ABB RobotStudio station: RoboX0.rspag

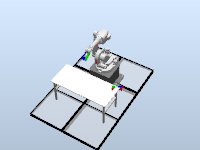
--- station ---
Station RoboX0 (saved by RobotStudio 21.3.9676.1)
Controller IRB1600_10_145, task T_ROB1: task frame (RAPID world) sits at (0, 0, 520) mm in the station
Controller IRB1600_10_145
  mechanical unit ROB_1: IRB1600_10_145__01_2, 6 joints, base frame (0, 0, 0) mm
Layout (positions relative to the parent item):
  - IRB1600_10_145__01_2 [mechanism, from Robots\IRB1600_10_145_G_01.rslib] at (0, 0, 520) mm; joint values [0, 0, 0, 0, 0.5236, 0] (rad or m)
  - подставка [part, from Libraries\box.rslib]
  - Стол сборка_4 [part, from Libraries\table.rslib] at (975, 0, 0) mm, rotated rx 0 ry 0 rz 90 deg
  - gripper2 [mechanism, from Libraries\gripper.rslib] at (806.29, 0, 1674) mm, rotated rx 180 ry 60 rz 180 deg; joint values [0] (rad or m)
Attachment: gripper2 is attached to IRB1600_10_145__01_2 / Link6

--- Backups/IRB1600_10_145/RAPID/TASK1/PROGMOD/CalibData.mod ---
MODULE CalibData
    TASK PERS wobjdata Workobject_1:=[FALSE,TRUE,"",[[606.263,790,210],[0.707106781,0,0,0.707106781]],[[-100,-100,0],[0,-0.707106781,0.707106781,0]]];
    PERS tooldata gripper:=[TRUE,[[0,0,115],[1,0,0,0]],[0.5,[0,0,30],[1,0,0,0],0,0,0]];
ENDMODULE

--- Backups/IRB1600_10_145/RAPID/TASK1/PROGMOD/Module1.mod ---
MODULE Module1
        CONST robtarget Target_10:=[[199.621572681,690,-886.5],[0,0.5,0,0.866025404],[0,0,0,0],[9E+09,9E+09,9E+09,9E+09,9E+09,9E+09]];

        CONST robtarget home:=[[199.621572681,690,-886.5],[0,0.5,0,0.866025404],[0,0,0,0],[9E+09,9E+09,9E+09,9E+09,9E+09,9E+09]];
        CONST robtarget storeX:=[[199.621572681,690,-886.5],[0,0.5,0,0.866025404],[0,0,0,0],[9E+09,9E+09,9E+09,9E+09,9E+09,9E+09]];
        CONST robtarget store0:=[[199.621572681,690,-886.5],[0,0.5,0,0.866025404],[0,0,0,0],[9E+09,9E+09,9E+09,9E+09,9E+09,9E+09]];
        CONST robtarget fieldCenter:=[[199.621572681,690,-886.5],[0,0.5,0,0.866025404],[0,0,0,0],[9E+09,9E+09,9E+09,9E+09,9E+09,9E+09]];

        CONST num zazor := 30;


        ! Player
        ! 1 - X
        ! 2 - 0
        ! 0 - game over
        PERS string PlayerStr := "0";
        VAR robtarget curStore;
        VAR num Player:=1;
        VAR num field{3,3}:=[
        [0,0,0],
        [0,0,0],
        [0,0,0]
        ];


        ! delta x To
        CONST num dxT :=0;
        CONST num dyT :=0;
        CONST num dzT :=0;


        CONST num ActStep:=1;
        CONST num ActEndGame:=3;
        CONST num ActWinGame:=4;

        PERS num Action:=1;

    PROC main()
        PlayerStr:="W";
        Action :=0;
        WHILE TRUE DO
            chooseAction Action;
        ENDWHILE
    ENDPROC

    PROC chooseAction(num Action)

        IF Action = ActStep THEN
            moveX0;
        ELSEIF Action = ActEndGame THEN
            moveJ home, v100, z100, gripper;
        ENDIF

        Action := 0;

    ENDPROC

    PROC moveX0()
        VAR num i := 2 + dxT/60;
        VAR num j := 4 -  2 + dyT/60;

        IF field{i,j}=0 THEN
            field{i,j} := Player;

            IF Player=0 OR Player=1 THEN
                curStore := storeX;
                Player:=2;
                PlayerStr:="0";
            ELSE
                curStore := store0;
                Player:=1;
                PlayerStr:="X";
            ENDIF

            moveCube curStore, Offs(fieldCenter, dXT,dyT, dzT);
        ENDIF
    ENDPROC

    PROC moveCube(robtarget pfrom, robtarget pto)
        grab(pfrom);
        stand(pto);
    ENDPROC

    PROC grab(robtarget point)
        MoveJ point,v1000,z1,gripper\WObj:=Workobject_1;
        MoveL Offs(point, 0,0,zazor),v100,fine,gripper\WObj:=Workobject_1;
        PulseDO\High,do_GripClose;

        !WaitDI di_GripClosed,1;
        MoveJ point,v100,z1,gripper\WObj:=Workobject_1;
    ENDPROC

    PROC stand(robtarget point)
        MoveJ point,v1000,z1,gripper\WObj:=Workobject_1;
        MoveL Offs(point, 0,0,zazor),v100,fine,gripper\WObj:=Workobject_1;
        PulseDO\High,do_GripOpen;
        !WaitDI di_GripOpened,1;
        MoveJ point,v100,z1,gripper\WObj:=Workobject_1;
    ENDPROC
    PROC Path_10()
        MoveL Target_10,v1000,z100,gripper\WObj:=Workobject_1;
    ENDPROC



ENDMODULE

--- Backups/IRB1600_10_145/SYSPAR/EIO.cfg ---
EIO:CFG_1.0:6:1::
#
EIO_SIGNAL:

      -Name "do_GripClose" -SignalType "DO"

      -Name "do_GripOpen" -SignalType "DO"

      -Name "di_GripOpened" -SignalType "DI"

      -Name "di_GripClosed" -SignalType "DI"
